(* Logix 5000 project; controller STAT 1756-L72 rev 20.12; software revision 20.04; part 4 of 34 *)
(* tags used below, declared in another part *)
   B3 : DINT[10];
   N20 : DINT[50];
   N7 : DINT[30];
   N9 : DINT[50];
   T4 : TIMER[25];
   DateTime : DINT[7];   // DINT array tag for retrieve wallclock time through GSV created during conversion
   def1bassin : DINT;
   def2bassin : DINT;
   p15 : BOOL;
   P16 : BOOL;
   P17 : BOOL;
   P18 : BOOL;
   P3 : BOOL;
   P4 : BOOL;
   S_FLOW_VENTURI : DINT;
   S_Lvl_incident_bak : DINT;
   S_PH_naar_venturi : DINT;
   S_Ph_Neutral : DINT;
   S_PH_venturi : DINT;
   S_pos_V_renv : DINT;
   s_pos_V_venturi_open : BOOL;
(* BASSIN, continued *)

ROUTINE _3_PMP   (* ladder *)
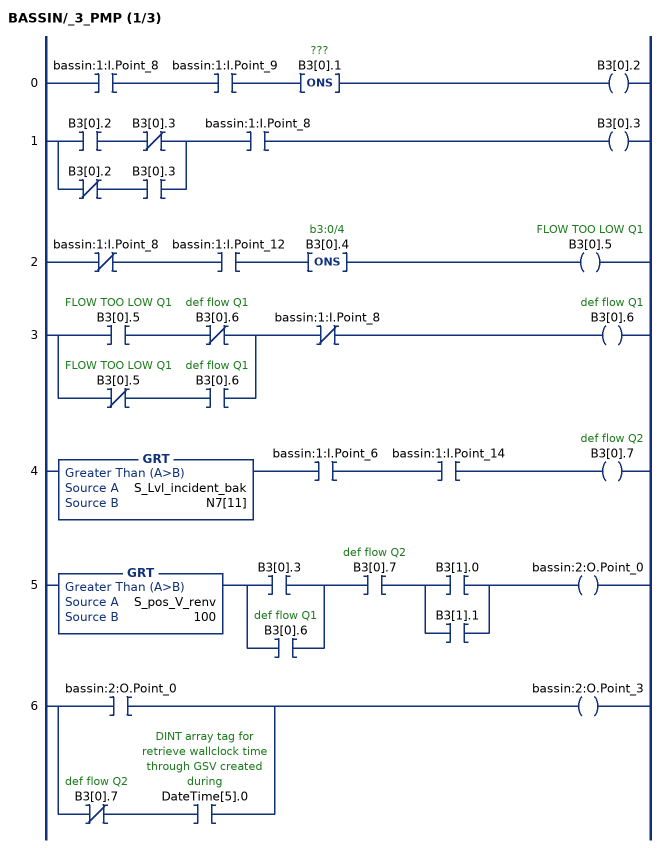
   0: XIC(bassin:1:I.Point_8)XIC(bassin:1:I.Point_9)ONS(B3[0].1)OTE(B3[0].2);
   1: [XIC(B3[0].2) XIO(B3[0].3) ,XIO(B3[0].2) XIC(B3[0].3) ]XIC(bassin:1:I.Point_8)OTE(B3[0].3);
   2: XIO(bassin:1:I.Point_8)XIC(bassin:1:I.Point_12)ONS(B3[0].4)OTE(B3[0].5);
   3: [XIC(B3[0].5) XIO(B3[0].6) ,XIO(B3[0].5) XIC(B3[0].6) ]XIO(bassin:1:I.Point_8)OTE(B3[0].6);
   4: GRT(S_Lvl_incident_bak,N7[11])XIC(bassin:1:I.Point_6)XIC(bassin:1:I.Point_14)OTE(B3[0].7);
   5: GRT(S_pos_V_renv,100)[XIC(B3[0].3) ,XIC(B3[0].6) ]XIC(B3[0].7)[XIC(B3[1].0) ,XIC(B3[1].1) ]OTE(bassin:2:O.Point_0);
   6: [XIC(bassin:2:O.Point_0) ,XIO(B3[0].7) XIC(DateTime[5].0) ]OTE(bassin:2:O.Point_3);
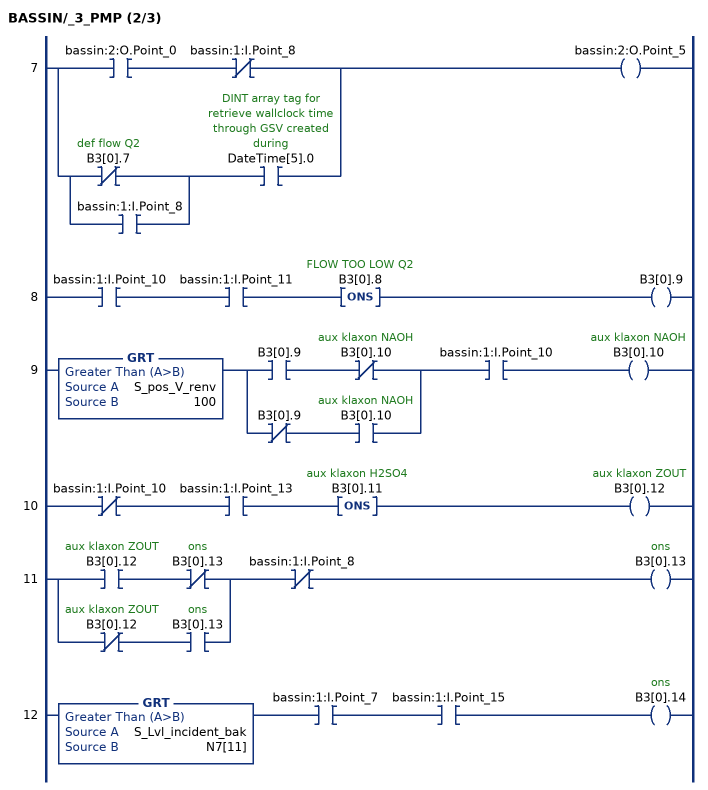
   7: [XIC(bassin:2:O.Point_0) XIO(bassin:1:I.Point_8) ,[XIO(B3[0].7) ,XIC(bassin:1:I.Point_8) ] XIC(DateTime[5].0) ]OTE(bassin:2:O.Point_5);
   8: XIC(bassin:1:I.Point_10)XIC(bassin:1:I.Point_11)ONS(B3[0].8)OTE(B3[0].9);
   9: GRT(S_pos_V_renv,100)[XIC(B3[0].9) XIO(B3[0].10) ,XIO(B3[0].9) XIC(B3[0].10) ]XIC(bassin:1:I.Point_10)OTE(B3[0].10);
   10: XIO(bassin:1:I.Point_10)XIC(bassin:1:I.Point_13)ONS(B3[0].11)OTE(B3[0].12);
   11: [XIC(B3[0].12) XIO(B3[0].13) ,XIO(B3[0].12) XIC(B3[0].13) ]XIO(bassin:1:I.Point_8)OTE(B3[0].13);
   12: GRT(S_Lvl_incident_bak,N7[11])XIC(bassin:1:I.Point_7)XIC(bassin:1:I.Point_15)OTE(B3[0].14);
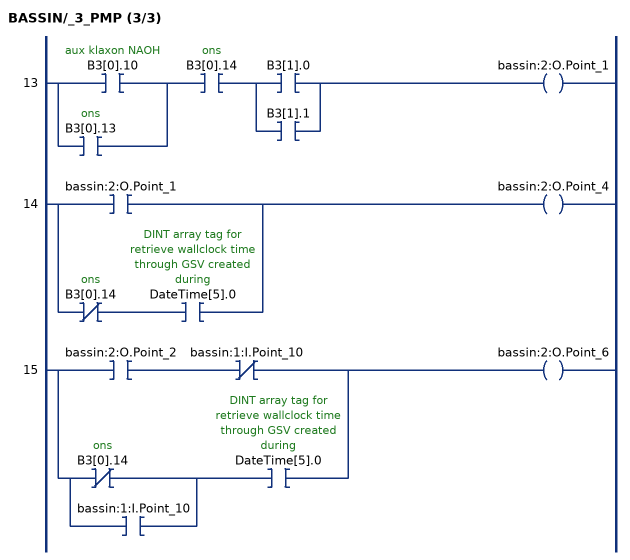
   13: [XIC(B3[0].10) ,XIC(B3[0].13) ]XIC(B3[0].14)[XIC(B3[1].0) ,XIC(B3[1].1) ]OTE(bassin:2:O.Point_1);
   14: [XIC(bassin:2:O.Point_1) ,XIO(B3[0].14) XIC(DateTime[5].0) ]OTE(bassin:2:O.Point_4);
   15: [XIC(bassin:2:O.Point_2) XIO(bassin:1:I.Point_10) ,[XIO(B3[0].14) ,XIC(bassin:1:I.Point_10) ] XIC(DateTime[5].0) ]OTE(bassin:2:O.Point_6);
END_ROUTINE

ROUTINE _4_VENTURI   (* ladder *)
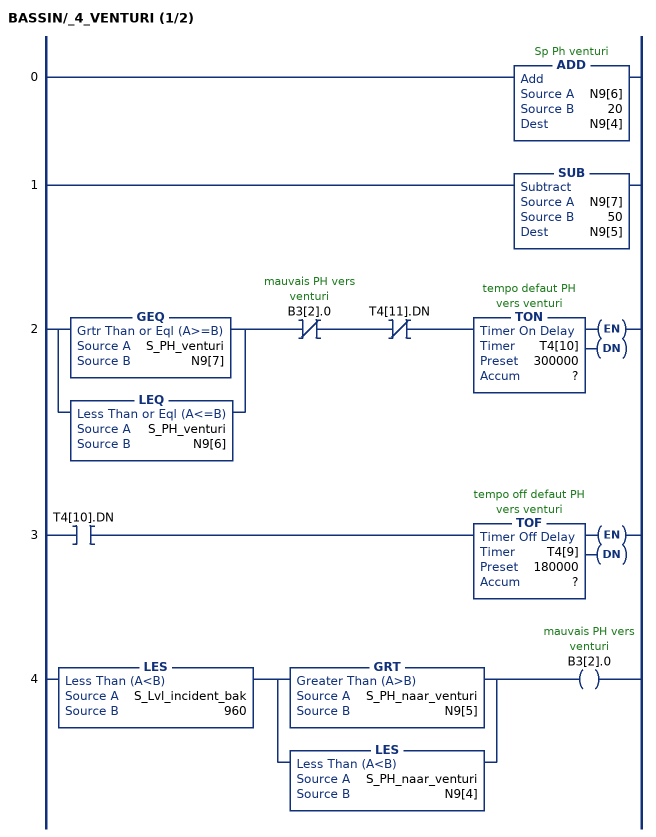
   0: ADD(N9[6],20,N9[4]);
   1: SUB(N9[7],50,N9[5]);
   2: [GEQ(S_PH_venturi,N9[7]) ,LEQ(S_PH_venturi,N9[6]) ]XIO(B3[2].0)XIO(T4[11].DN)TON(T4[10],?,?);
   3: XIC(T4[10].DN)TOF(T4[9],?,?);
   4: LES(S_Lvl_incident_bak,960)[GRT(S_PH_naar_venturi,N9[5]) ,LES(S_PH_naar_venturi,N9[4]) ]OTE(B3[2].0);
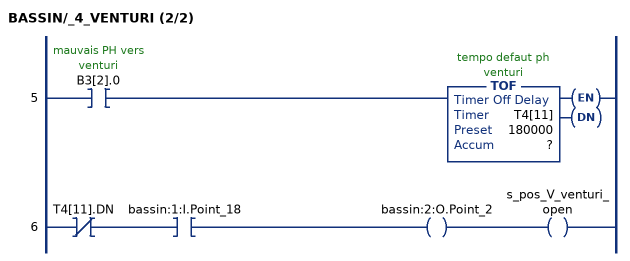
   5: XIC(B3[2].0)TOF(T4[11],?,?);
   6: XIO(T4[11].DN)XIC(bassin:1:I.Point_18)OTE(bassin:2:O.Point_2)OTE(s_pos_V_venturi_open);
END_ROUTINE

ROUTINE _5_REGUL_PH   (* ladder *)
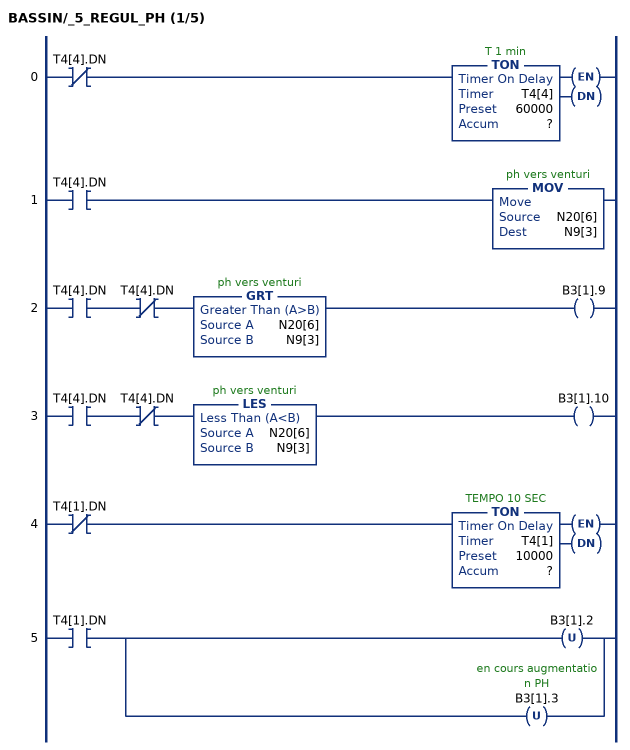
   0: XIO(T4[4].DN)TON(T4[4],?,?);
   1: XIC(T4[4].DN)MOV(N20[6],N9[3]);
   2: XIC(T4[4].DN)XIO(T4[4].DN)GRT(N20[6],N9[3])OTE(B3[1].9);
   3: XIC(T4[4].DN)XIO(T4[4].DN)LES(N20[6],N9[3])OTE(B3[1].10);
   4: XIO(T4[1].DN)TON(T4[1],?,?);
   5: XIC(T4[1].DN)[OTU(B3[1].2) ,OTU(B3[1].3) ];
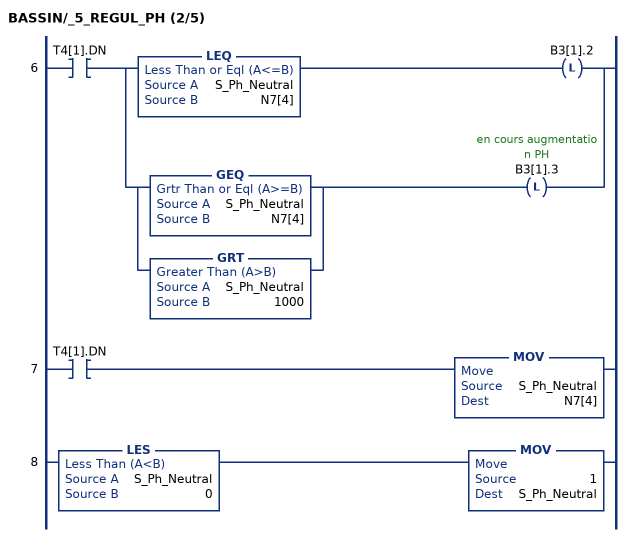
   6: XIC(T4[1].DN)[LEQ(S_Ph_Neutral,N7[4]) OTL(B3[1].2) ,[GEQ(S_Ph_Neutral,N7[4]) ,GRT(S_Ph_Neutral,1000) ] OTL(B3[1].3) ];
   7: XIC(T4[1].DN)MOV(S_Ph_Neutral,N7[4]);
   8: LES(S_Ph_Neutral,0)MOV(1,S_Ph_Neutral);
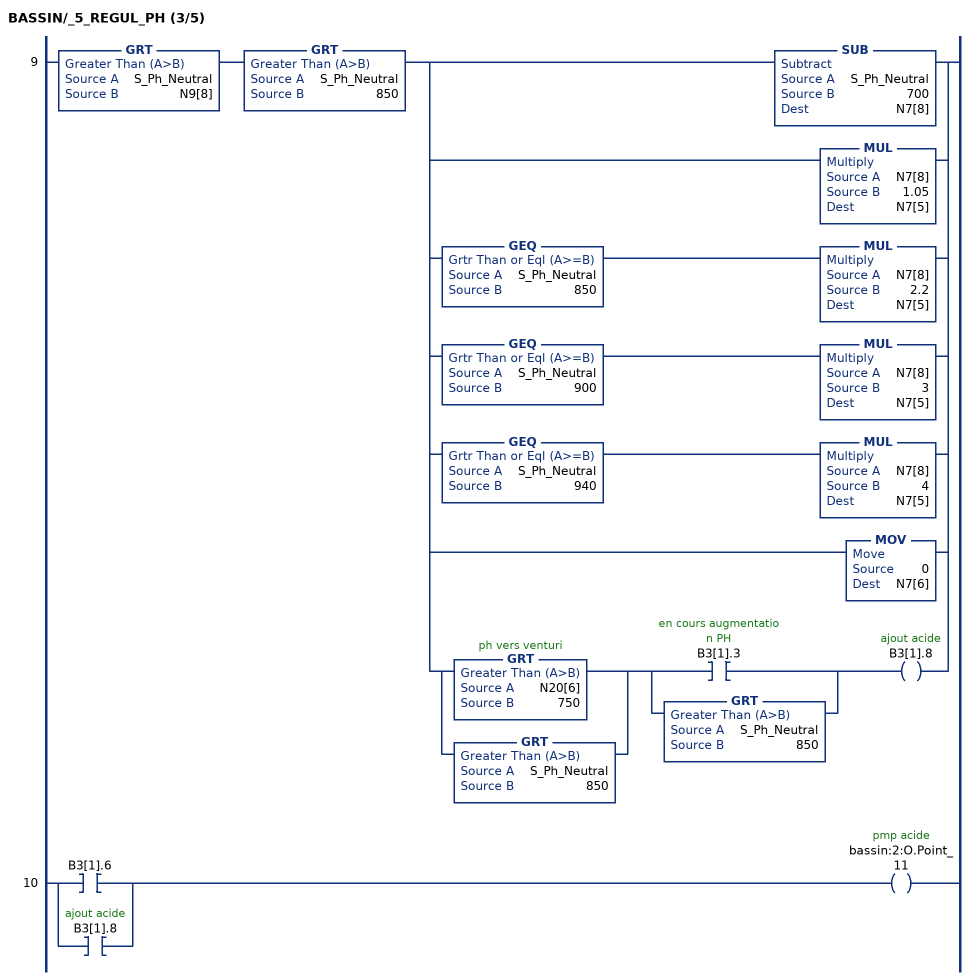
   9: GRT(S_Ph_Neutral,N9[8])GRT(S_Ph_Neutral,850)[SUB(S_Ph_Neutral,700,N7[8]) ,MUL(N7[8],1.05,N7[5]) ,GEQ(S_Ph_Neutral,850) MUL(N7[8],2.2,N7[5]) ,GEQ(S_Ph_Neutral,900) MUL(N7[8],3,N7[5]) ,GEQ(S_Ph_Neutral,940) MUL(N7[8],4,N7[5]) ,MOV(0,N7[6]) ,[GRT(N20[6],750) ,GRT(S_Ph_Neutral,850) ] [XIC(B3[1].3) ,GRT(S_Ph_Neutral,850) ] OTE(B3[1].8) ];
   10: [XIC(B3[1].6) ,XIC(B3[1].8) ]OTE(bassin:2:O.Point_11);
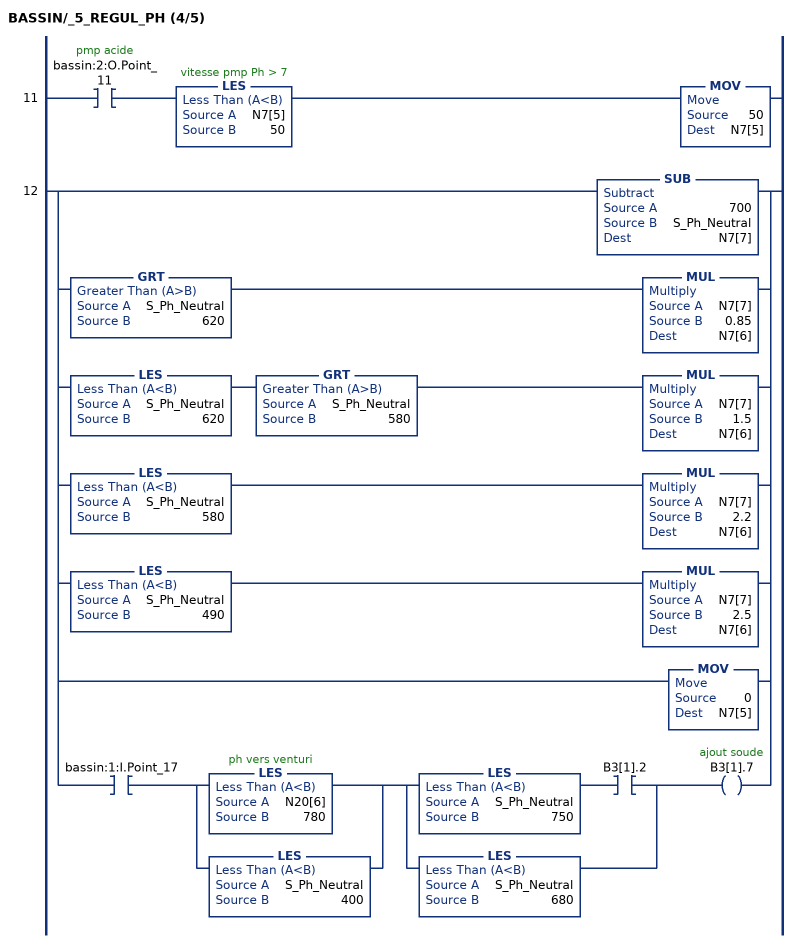
   11: XIC(bassin:2:O.Point_11)LES(N7[5],50)MOV(50,N7[5]);
   12: [SUB(700,S_Ph_Neutral,N7[7]) ,GRT(S_Ph_Neutral,620) MUL(N7[7],0.85,N7[6]) ,LES(S_Ph_Neutral,620) GRT(S_Ph_Neutral,580) MUL(N7[7],1.5,N7[6]) ,LES(S_Ph_Neutral,580) MUL(N7[7],2.2,N7[6]) ,LES(S_Ph_Neutral,490) MUL(N7[7],2.5,N7[6]) ,MOV(0,N7[5]) ,XIC(bassin:1:I.Point_17) [LES(N20[6],780) ,LES(S_Ph_Neutral,400) ] [LES(S_Ph_Neutral,750) XIC(B3[1].2) ,LES(S_Ph_Neutral,680) ] OTE(B3[1].7) ];
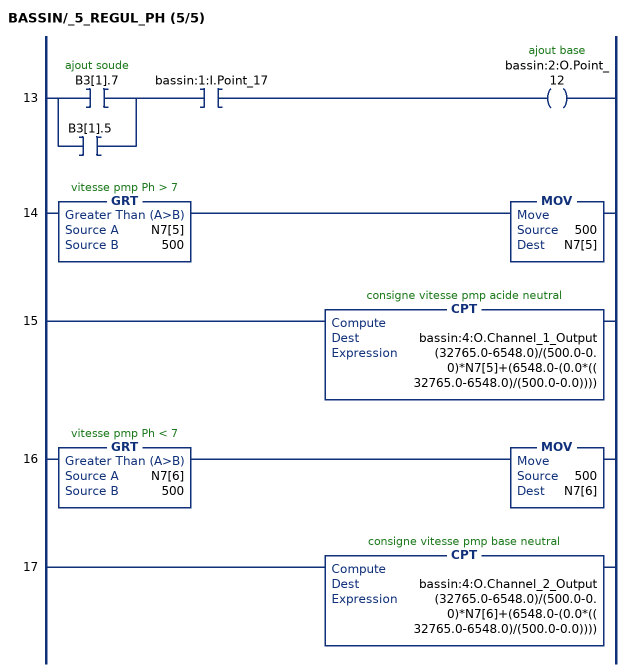
   13: [XIC(B3[1].7) ,XIC(B3[1].5) ]XIC(bassin:1:I.Point_17)OTE(bassin:2:O.Point_12);
   14: GRT(N7[5],500)MOV(500,N7[5]);
   15: CPT(bassin:4:O.Channel_1_Output,(32765.0-6548.0)/(500.0-0.0)*N7[5]+(6548.0-(0.0*((32765.0-6548.0)/(500.0-0.0)))));
   16: GRT(N7[6],500)MOV(500,N7[6]);
   17: CPT(bassin:4:O.Channel_2_Output,(32765.0-6548.0)/(500.0-0.0)*N7[6]+(6548.0-(0.0*((32765.0-6548.0)/(500.0-0.0)))));
END_ROUTINE

ROUTINE _6_ALARM   (* ladder *)
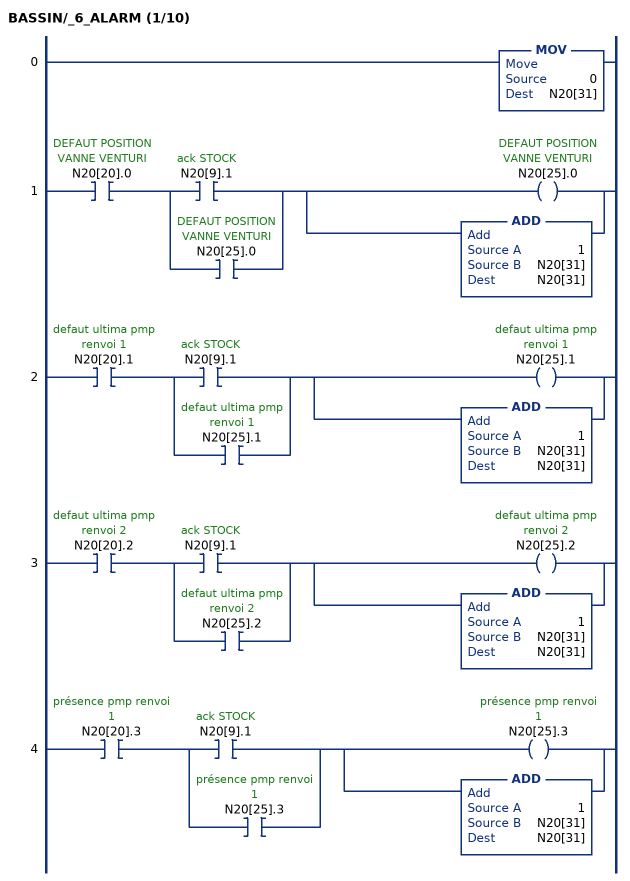
   0: MOV(0,N20[31]);
   1: XIC(N20[20].0)[XIC(N20[9].1) ,XIC(N20[25].0) ][OTE(N20[25].0) ,ADD(1,N20[31],N20[31]) ];
   2: XIC(N20[20].1)[XIC(N20[9].1) ,XIC(N20[25].1) ][OTE(N20[25].1) ,ADD(1,N20[31],N20[31]) ];
   3: XIC(N20[20].2)[XIC(N20[9].1) ,XIC(N20[25].2) ][OTE(N20[25].2) ,ADD(1,N20[31],N20[31]) ];
   4: XIC(N20[20].3)[XIC(N20[9].1) ,XIC(N20[25].3) ][OTE(N20[25].3) ,ADD(1,N20[31],N20[31]) ];
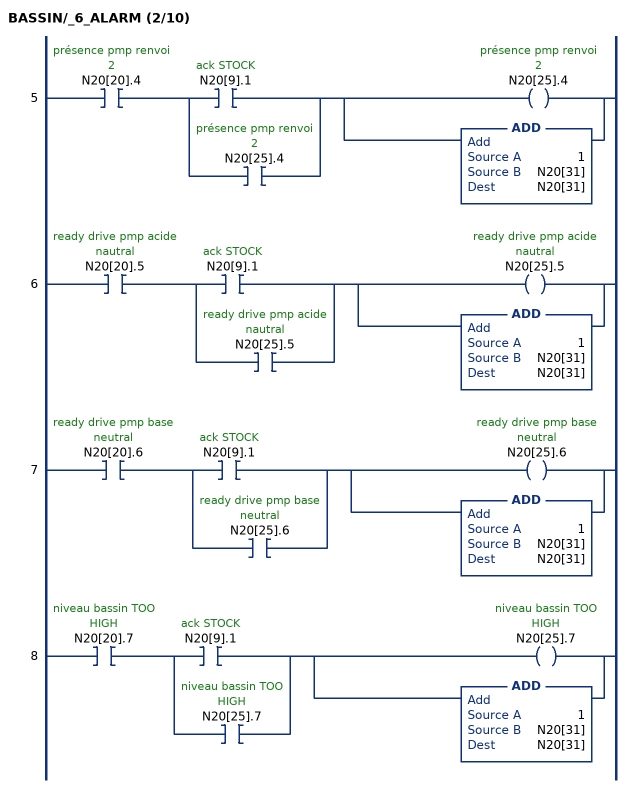
   5: XIC(N20[20].4)[XIC(N20[9].1) ,XIC(N20[25].4) ][OTE(N20[25].4) ,ADD(1,N20[31],N20[31]) ];
   6: XIC(N20[20].5)[XIC(N20[9].1) ,XIC(N20[25].5) ][OTE(N20[25].5) ,ADD(1,N20[31],N20[31]) ];
   7: XIC(N20[20].6)[XIC(N20[9].1) ,XIC(N20[25].6) ][OTE(N20[25].6) ,ADD(1,N20[31],N20[31]) ];
   8: XIC(N20[20].7)[XIC(N20[9].1) ,XIC(N20[25].7) ][OTE(N20[25].7) ,ADD(1,N20[31],N20[31]) ];
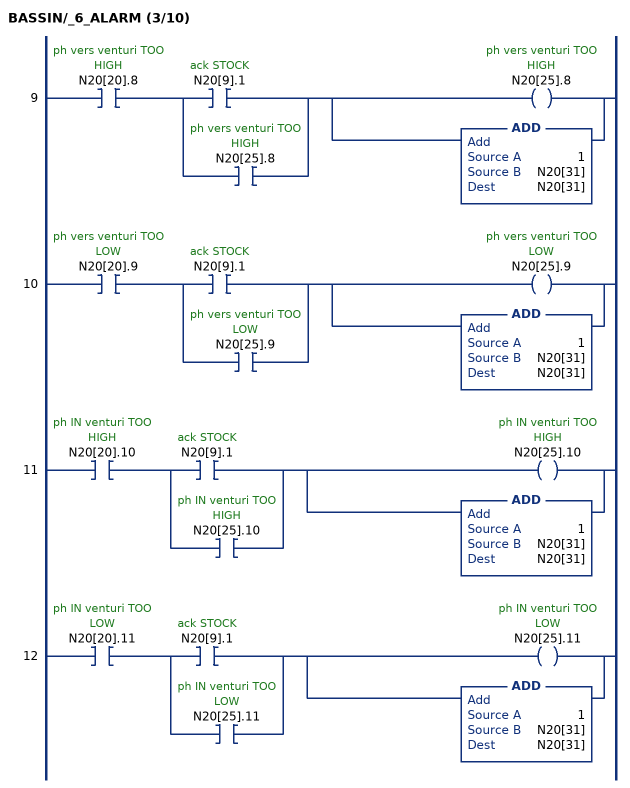
   9: XIC(N20[20].8)[XIC(N20[9].1) ,XIC(N20[25].8) ][OTE(N20[25].8) ,ADD(1,N20[31],N20[31]) ];
   10: XIC(N20[20].9)[XIC(N20[9].1) ,XIC(N20[25].9) ][OTE(N20[25].9) ,ADD(1,N20[31],N20[31]) ];
   11: XIC(N20[20].10)[XIC(N20[9].1) ,XIC(N20[25].10) ][OTE(N20[25].10) ,ADD(1,N20[31],N20[31]) ];
   12: XIC(N20[20].11)[XIC(N20[9].1) ,XIC(N20[25].11) ][OTE(N20[25].11) ,ADD(1,N20[31],N20[31]) ];
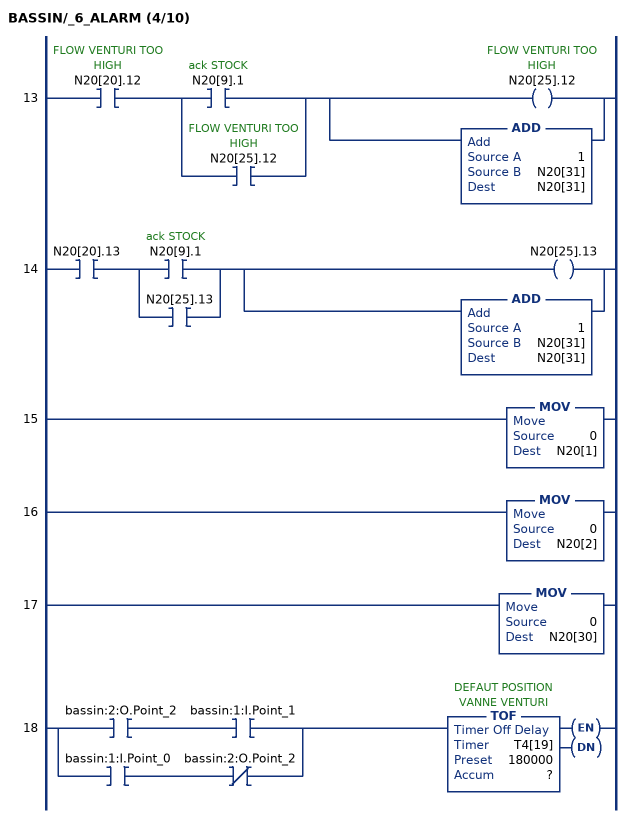
   13: XIC(N20[20].12)[XIC(N20[9].1) ,XIC(N20[25].12) ][OTE(N20[25].12) ,ADD(1,N20[31],N20[31]) ];
   14: XIC(N20[20].13)[XIC(N20[9].1) ,XIC(N20[25].13) ][OTE(N20[25].13) ,ADD(1,N20[31],N20[31]) ];
   15: MOV(0,N20[1]);
   16: MOV(0,N20[2]);
   17: MOV(0,N20[30]);
   18: [XIC(bassin:2:O.Point_2) XIC(bassin:1:I.Point_1) ,XIC(bassin:1:I.Point_0) XIO(bassin:2:O.Point_2) ]TOF(T4[19],?,?);
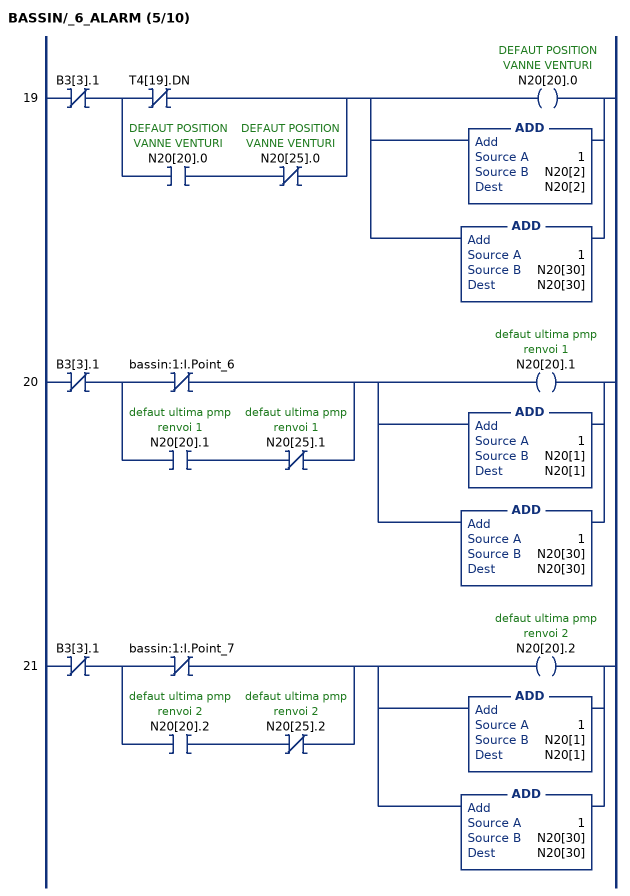
   19: XIO(B3[3].1)[XIO(T4[19].DN) ,XIC(N20[20].0) XIO(N20[25].0) ][OTE(N20[20].0) ,ADD(1,N20[2],N20[2]) ,ADD(1,N20[30],N20[30]) ];
   20: XIO(B3[3].1)[XIO(bassin:1:I.Point_6) ,XIC(N20[20].1) XIO(N20[25].1) ][OTE(N20[20].1) ,ADD(1,N20[1],N20[1]) ,ADD(1,N20[30],N20[30]) ];
   21: XIO(B3[3].1)[XIO(bassin:1:I.Point_7) ,XIC(N20[20].2) XIO(N20[25].2) ][OTE(N20[20].2) ,ADD(1,N20[1],N20[1]) ,ADD(1,N20[30],N20[30]) ];
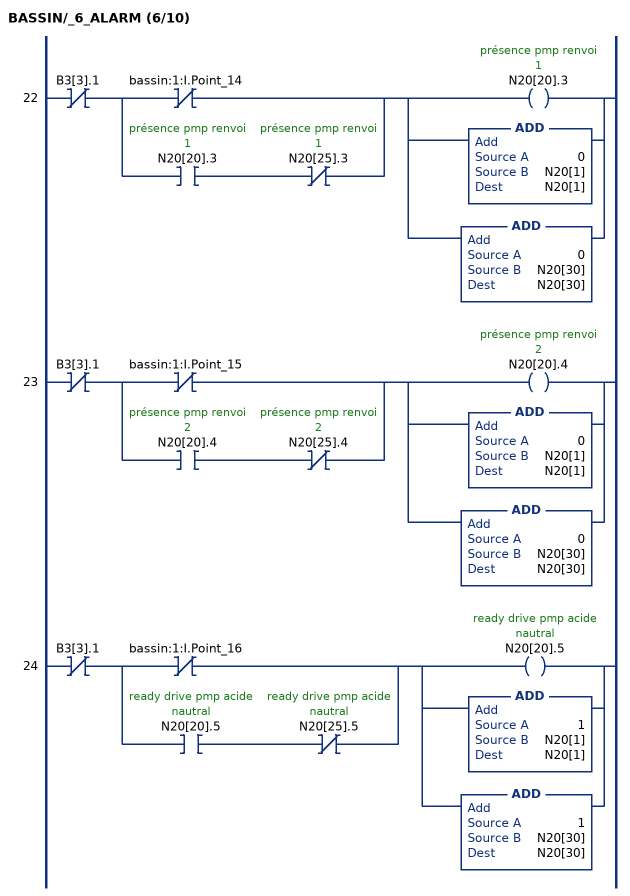
   22: XIO(B3[3].1)[XIO(bassin:1:I.Point_14) ,XIC(N20[20].3) XIO(N20[25].3) ][OTE(N20[20].3) ,ADD(0,N20[1],N20[1]) ,ADD(0,N20[30],N20[30]) ];
   23: XIO(B3[3].1)[XIO(bassin:1:I.Point_15) ,XIC(N20[20].4) XIO(N20[25].4) ][OTE(N20[20].4) ,ADD(0,N20[1],N20[1]) ,ADD(0,N20[30],N20[30]) ];
   24: XIO(B3[3].1)[XIO(bassin:1:I.Point_16) ,XIC(N20[20].5) XIO(N20[25].5) ][OTE(N20[20].5) ,ADD(1,N20[1],N20[1]) ,ADD(1,N20[30],N20[30]) ];
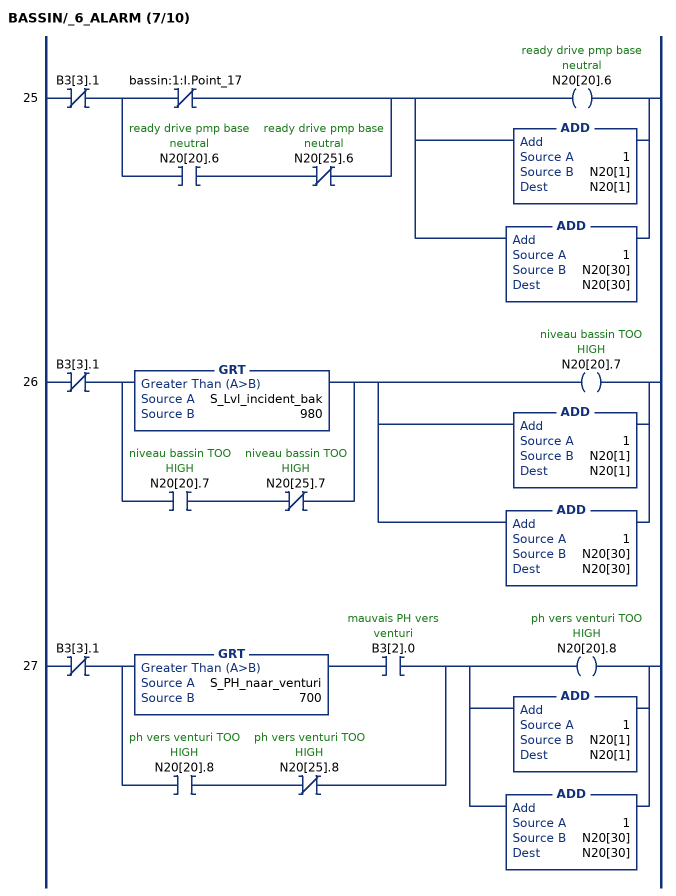
   25: XIO(B3[3].1)[XIO(bassin:1:I.Point_17) ,XIC(N20[20].6) XIO(N20[25].6) ][OTE(N20[20].6) ,ADD(1,N20[1],N20[1]) ,ADD(1,N20[30],N20[30]) ];
   26: XIO(B3[3].1)[GRT(S_Lvl_incident_bak,980) ,XIC(N20[20].7) XIO(N20[25].7) ][OTE(N20[20].7) ,ADD(1,N20[1],N20[1]) ,ADD(1,N20[30],N20[30]) ];
   27: XIO(B3[3].1)[GRT(S_PH_naar_venturi,700) XIC(B3[2].0) ,XIC(N20[20].8) XIO(N20[25].8) ][OTE(N20[20].8) ,ADD(1,N20[1],N20[1]) ,ADD(1,N20[30],N20[30]) ];
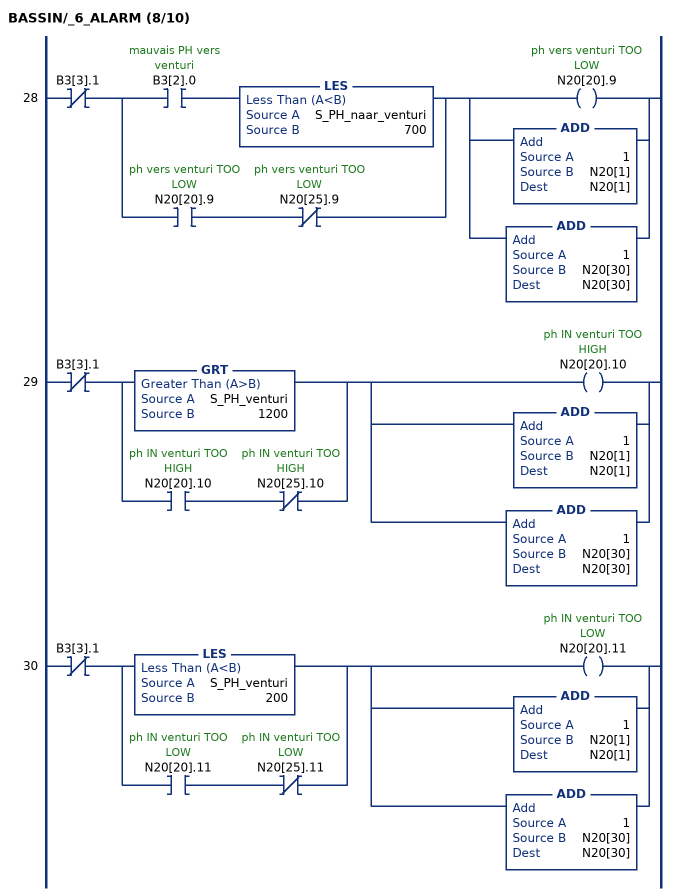
   28: XIO(B3[3].1)[XIC(B3[2].0) LES(S_PH_naar_venturi,700) ,XIC(N20[20].9) XIO(N20[25].9) ][OTE(N20[20].9) ,ADD(1,N20[1],N20[1]) ,ADD(1,N20[30],N20[30]) ];
   29: XIO(B3[3].1)[GRT(S_PH_venturi,1200) ,XIC(N20[20].10) XIO(N20[25].10) ][OTE(N20[20].10) ,ADD(1,N20[1],N20[1]) ,ADD(1,N20[30],N20[30]) ];
   30: XIO(B3[3].1)[LES(S_PH_venturi,200) ,XIC(N20[20].11) XIO(N20[25].11) ][OTE(N20[20].11) ,ADD(1,N20[1],N20[1]) ,ADD(1,N20[30],N20[30]) ];
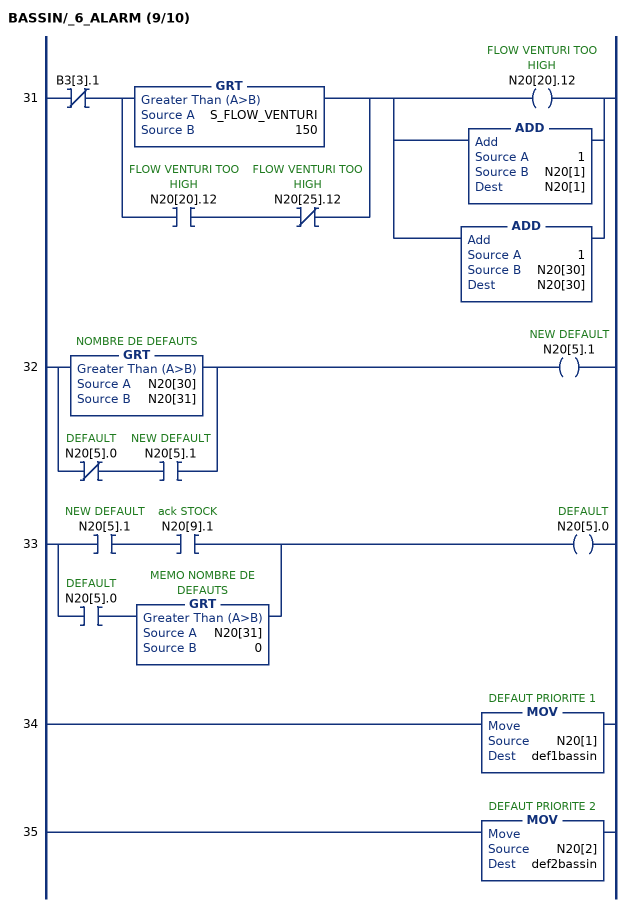
   31: XIO(B3[3].1)[GRT(S_FLOW_VENTURI,150) ,XIC(N20[20].12) XIO(N20[25].12) ][OTE(N20[20].12) ,ADD(1,N20[1],N20[1]) ,ADD(1,N20[30],N20[30]) ];
   32: [GRT(N20[30],N20[31]) ,XIO(N20[5].0) XIC(N20[5].1) ]OTE(N20[5].1);
   33: [XIC(N20[5].1) XIC(N20[9].1) ,XIC(N20[5].0) GRT(N20[31],0) ]OTE(N20[5].0);
   34: MOV(N20[1],def1bassin);
   35: MOV(N20[2],def2bassin);
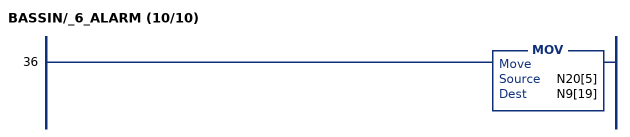
   36: MOV(N20[5],N9[19]);
END_ROUTINE
